(* Logix 5000 project; controller PLC_253_Base vendor 1 type 14 code 156 rev 30.11; software revision 30.00 *)

TASK MainTask (continuous, watchdog 500 ms) : MainProgram

MODULES
   Local : vendor 1 type 14 code 156 (Compact 0, rev 30.11)
      DI_4 : 1769-IQ16 (Compact 4, rev 1.1, Input RPI 20 ms)
      DO_5 : vendor 1 type 7 code 86 (Compact 5, rev 2.1, Output RPI 20 ms)
END_MODULES

VAR_GLOBAL   (* controller tags *)
   Count_S1 : COUNTER := (PRE := 3);
   FS_BANDA1 : ALIAS FOR Local:5:O.Data.0;
   FS_START : ALIAS FOR Local:4:I.Data.1;
   FS_STOP : ALIAS FOR Local:4:I.Data.0;
   GD_IN_0 : BOOL := 1;
   GD_IN_1 : BOOL;
   GD_IN_2 : BOOL;   // GD Sensor1
   GD_IN_3 : BOOL := 1;
   GD_IN_4 : BOOL := 1;
   GD_IN_5 : BOOL;   // GD Reset
   GD_OUT_0 : BOOL;
   GD_OUT_1 : BOOL;
   GD_OUT_2 : BOOL := 1;
   TagA : BOOL;
   Timer1 : TIMER := (PRE := 5000);
   VarX : BOOL;
END_VAR

PROGRAM MainProgram   (* main routine MainRoutine *)

ROUTINE MainRoutine   (* ladder *)
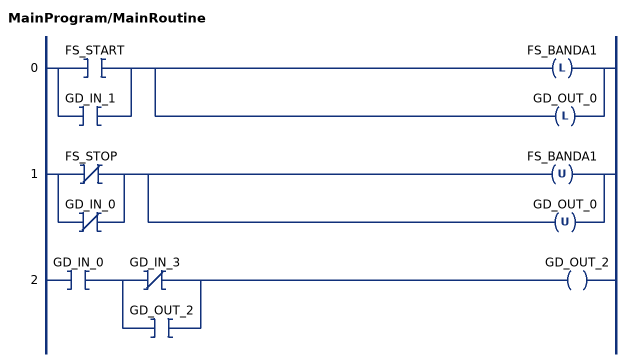
   0: [XIC(FS_START) ,XIC(GD_IN_1) ][OTL(FS_BANDA1) ,OTL(GD_OUT_0) ];
   1: [XIO(FS_STOP) ,XIO(GD_IN_0) ][OTU(FS_BANDA1) ,OTU(GD_OUT_0) ];
   2: XIC(GD_IN_0)[XIO(GD_IN_3) ,XIC(GD_OUT_2) ]OTE(GD_OUT_2);
END_ROUTINE
END_PROGRAM
